INTERFACE I_QueueItem EXTENDS I_LinkedListItem_ReadWrite

END_INTERFACE

(* stored: Version 1.1.0.1, ProductVersion 3.1.4024.12
   Itf I_QueueItem: Id {21205a69-1823-4afb-90bd-73670b0f507d} *)
